{attribute 'GeneratedUsingTerminal: AT2025-0250-0020'}
{attribute addProperty BoxType "AT2025-0250-0020"}
{attribute addProperty Id "A_0074_AT2000_5250_0017_AT2000_5250AT2000_01D6DEDF80"}
{attribute addProperty CRC "523179924"}
{attribute addProperty Size "80"}
TYPE A_0062_AT2025_0250_0020_AT2025_0250_1F2F1794 EXTENDS AT2025_86175B41 :
STRUCT
	{attribute addProperty Name "A_0074_AT2000_5250_0017_AT2000_5250"}
	A_0074_AT2000_5250_0017_AT2000_5250 : AT2000_01D6DEDF;
END_STRUCT
END_TYPE

(* stored: Version 1.2.0.0, ProductVersion 3.1.4024.9
   DUT A_0062_AT2025_0250_0020_AT2025_0250_1F2F1794: Id {75f0a2d5-dce3-4f8f-9a3c-99ce07a59680} *)
